PROGRAM MAIN
VAR
END_VAR

END_PROGRAM

(* stored: Version 1.1.0.1
   POU MAIN: Id {0ad4954e-ac64-46bb-9eb0-a0f0715ea3b1} *)
